KUKA KRL program: puntos.src, puntos.dat

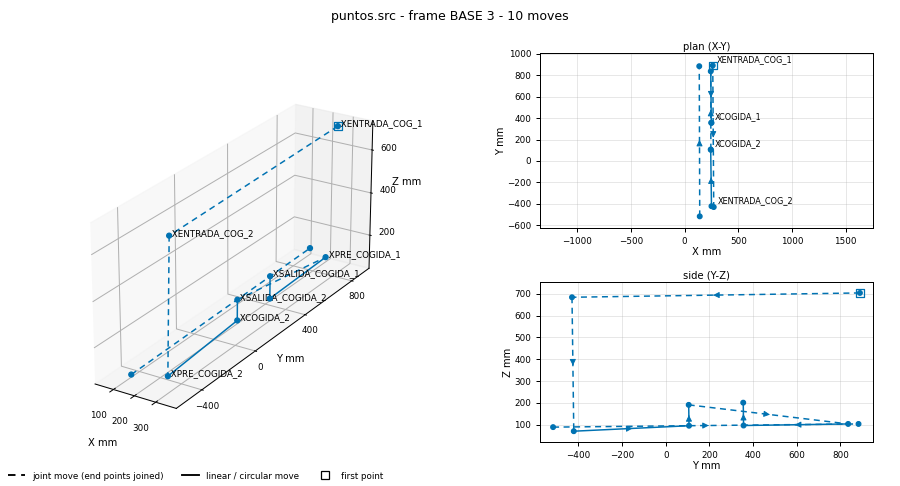
[picture p0: tool path of puntos.src in frame BASE 3, 10 of 13 moves have a stored position in this frame; points joined in program order, loops and branches not executed]
--- puntos.src ---
&ACCESS RVP
&REL 25
&PARAM TEMPLATE = C:\KRC\Roboter\Template\vorgabe
&PARAM EDITMASK = *
DEF PUNTOS( )
;FOLD INI
  ;FOLD BASISTECH INI
    GLOBAL INTERRUPT DECL 3 WHEN $STOPMESS==TRUE DO IR_STOPM ( )
    INTERRUPT ON 3
    BAS (#INITMOV,0 )
  ;ENDFOLD (BASISTECH INI)
  ;FOLD USER INI
    ;Make your modifications here

  ;ENDFOLD (USER INI)
;ENDFOLD (INI)


;FOLD PTP HOME Vel=100 % PDAT6;%{PE}%R 5.6.16,%MKUKATPBASIS,%CMOVE,%VPTP,%P 1:PTP, 2:HOME, 3:, 5:100, 7:PDAT6
$BWDSTART=FALSE
PDAT_ACT=PPDAT6
FDAT_ACT=FHOME
BAS(#PTP_PARAMS,100)
$H_POS=XHOME
PTP XHOME
;ENDFOLD


;FOLD PTP ENTRADA_COG_1 Vel=100 % PDAT1 Tool[2]:MORDAZA Base[3]:TRANSPORTADOR;%{PE}%R 5.6.16,%MKUKATPBASIS,%CMOVE,%VPTP,%P 1:PTP, 2:ENTRADA_COG_1, 3:, 5:100, 7:PDAT1
$BWDSTART=FALSE
PDAT_ACT=PPDAT1
FDAT_ACT=FENTRADA_COG_1
BAS(#PTP_PARAMS,100)
PTP XENTRADA_COG_1
;ENDFOLD


;FOLD PTP ENTRADA_COG_2 Vel=100 % PDAT2 Tool[2]:MORDAZA Base[3]:TRANSPORTADOR;%{PE}%R 5.6.16,%MKUKATPBASIS,%CMOVE,%VPTP,%P 1:PTP, 2:ENTRADA_COG_2, 3:, 5:100, 7:PDAT2
$BWDSTART=FALSE
PDAT_ACT=PPDAT2
FDAT_ACT=FENTRADA_COG_2
BAS(#PTP_PARAMS,100)
PTP XENTRADA_COG_2
;ENDFOLD


;FOLD PTP PRE_COGIDA_2 Vel=100 % PDAT3 Tool[2]:MORDAZA Base[3]:TRANSPORTADOR;%{PE}%R 5.6.16,%MKUKATPBASIS,%CMOVE,%VPTP,%P 1:PTP, 2:PRE_COGIDA_2, 3:, 5:100, 7:PDAT3
$BWDSTART=FALSE
PDAT_ACT=PPDAT3
FDAT_ACT=FPRE_COGIDA_2
BAS(#PTP_PARAMS,100)
PTP XPRE_COGIDA_2
;ENDFOLD


;FOLD LIN COGIDA_2 Vel=2 m/s CPDAT1 Tool[2]:MORDAZA Base[3]:TRANSPORTADOR;%{PE}%R 5.6.16,%MKUKATPBASIS,%CMOVE,%VLIN,%P 1:LIN, 2:COGIDA_2, 3:, 5:2, 7:CPDAT1
$BWDSTART=FALSE
LDAT_ACT=LCPDAT1
FDAT_ACT=FCOGIDA_2
BAS(#CP_PARAMS,2)
LIN XCOGIDA_2
;ENDFOLD


;FOLD LIN SALIDA_COGIDA_2 Vel=2 m/s CPDAT2 Tool[2]:MORDAZA Base[3]:TRANSPORTADOR;%{PE}%R 5.6.16,%MKUKATPBASIS,%CMOVE,%VLIN,%P 1:LIN, 2:SALIDA_COGIDA_2, 3:, 5:2, 7:CPDAT2
$BWDSTART=FALSE
LDAT_ACT=LCPDAT2
FDAT_ACT=FSALIDA_COGIDA_2
BAS(#CP_PARAMS,2)
LIN XSALIDA_COGIDA_2
;ENDFOLD



;FOLD PTP PRE_COGIDA_1 Vel=100 % PDAT4 Tool[2]:MORDAZA Base[3]:TRANSPORTADOR;%{PE}%R 5.6.16,%MKUKATPBASIS,%CMOVE,%VPTP,%P 1:PTP, 2:PRE_COGIDA_1, 3:, 5:100, 7:PDAT4
$BWDSTART=FALSE
PDAT_ACT=PPDAT4
FDAT_ACT=FPRE_COGIDA_1
BAS(#PTP_PARAMS,100)
PTP XPRE_COGIDA_1
;ENDFOLD


;FOLD LIN COGIDA_1 Vel=2 m/s CPDAT3 Tool[2]:MORDAZA Base[3]:TRANSPORTADOR;%{PE}%R 5.6.16,%MKUKATPBASIS,%CMOVE,%VLIN,%P 1:LIN, 2:COGIDA_1, 3:, 5:2, 7:CPDAT3
$BWDSTART=FALSE
LDAT_ACT=LCPDAT3
FDAT_ACT=FCOGIDA_1
BAS(#CP_PARAMS,2)
LIN XCOGIDA_1
;ENDFOLD


;FOLD LIN SALIDA_COGIDA_1 Vel=2 m/s CPDAT4 Tool[2]:MORDAZA Base[3]:TRANSPORTADOR;%{PE}%R 5.6.16,%MKUKATPBASIS,%CMOVE,%VLIN,%P 1:LIN, 2:SALIDA_COGIDA_1, 3:, 5:2, 7:CPDAT4
$BWDSTART=FALSE
LDAT_ACT=LCPDAT4
FDAT_ACT=FSALIDA_COGIDA_1
BAS(#CP_PARAMS,2)
LIN XSALIDA_COGIDA_1
;ENDFOLD



;FOLD PTP DEJA_DARSENA_2 Vel=100 % PDAT7 Tool[2]:MORDAZA Base[2]:DARSENA1;%{PE}%R 5.6.16,%MKUKATPBASIS,%CMOVE,%VPTP,%P 1:PTP, 2:DEJA_DARSENA_2, 3:, 5:100, 7:PDAT7
$BWDSTART=FALSE
PDAT_ACT=PPDAT7
FDAT_ACT=FDEJA_DARSENA_2
BAS(#PTP_PARAMS,100)
PTP XDEJA_DARSENA_2
;ENDFOLD


;FOLD PTP DEJA_DARSENA_1 Vel=100 % PDAT8 Tool[2]:MORDAZA Base[1]:DARSENA1;%{PE}%R 5.6.16,%MKUKATPBASIS,%CMOVE,%VPTP,%P 1:PTP, 2:DEJA_DARSENA_1, 3:, 5:100, 7:PDAT8
$BWDSTART=FALSE
PDAT_ACT=PPDAT8
FDAT_ACT=FDEJA_DARSENA_1
BAS(#PTP_PARAMS,100)
PTP XDEJA_DARSENA_1
;ENDFOLD


;FOLD PTP cog_desplazada Vel=100 % PDAT9 Tool[2]:MORDAZA Base[3]:TRANSPORTADOR;%{PE}%R 5.6.16,%MKUKATPBASIS,%CMOVE,%VPTP,%P 1:PTP, 2:cog_desplazada, 3:, 5:100, 7:PDAT9
$BWDSTART=FALSE
PDAT_ACT=PPDAT9
FDAT_ACT=Fcog_desplazada
BAS(#PTP_PARAMS,100)
PTP Xcog_desplazada
;ENDFOLD

;FOLD PTP cog_desplazada1 Vel=100 % PDAT10 Tool[2]:MORDAZA Base[3]:TRANSPORTADOR;%{PE}%R 5.6.16,%MKUKATPBASIS,%CMOVE,%VPTP,%P 1:PTP, 2:cog_desplazada1, 3:, 5:100, 7:PDAT10
$BWDSTART=FALSE
PDAT_ACT=PPDAT10
FDAT_ACT=Fcog_desplazada1
BAS(#PTP_PARAMS,100)
PTP Xcog_desplazada1
;ENDFOLD
END

--- puntos.dat ---
&ACCESS RVP
&REL 25
&PARAM TEMPLATE = C:\KRC\Roboter\Template\vorgabe
&PARAM EDITMASK = *
DEFDAT  PUNTOS
;FOLD EXTERNAL DECLARATIONS;%{PE}%MKUKATPBASIS,%CEXT,%VCOMMON,%P
;FOLD BASISTECH EXT;%{PE}%MKUKATPBASIS,%CEXT,%VEXT,%P
EXT  BAS (BAS_COMMAND  :IN,REAL  :IN )
DECL INT SUCCESS
;ENDFOLD (BASISTECH EXT)
;FOLD USER EXT;%{E}%MKUKATPUSER,%CEXT,%VEXT,%P
;Make here your modifications

;ENDFOLD (USER EXT)
;ENDFOLD (EXTERNAL DECLARATIONS)
DECL BASIS_SUGG_T LAST_BASIS={POINT1[] "cog_desplazada1         ",POINT2[] "cog_desplazada1         ",CP_PARAMS[] "CPDAT3                  ",PTP_PARAMS[] "PDAT10                  ",CONT[] "                        ",CP_VEL[] "2                       ",PTP_VEL[] "100                     ",SYNC_PARAMS[] "SYNCDAT                 ",SPL_NAME[] "S0                      "}
DECL INT LAST_XP_POINT=0
DECL E6POS XP1={X 267.31131,Y 380.834595,Z 696.146973,A 1.043558,B 1.65328801,C 179.309006,S 6,T 59,E1 0.0,E2 0.0,E3 0.0,E4 0.0,E5 0.0,E6 0.0}
DECL FDAT FP1={TOOL_NO 2,BASE_NO 3,IPO_FRAME #BASE,POINT2[] " ",TQ_STATE FALSE}
DECL PDAT PPDAT1={VEL 100.0,ACC 100.0,APO_DIST 100.0}
DECL E6POS XENTRADA_COG_1={X 262.194702,Y 889.154297,Z 703.763123,A 1.04380703,B 1.65313005,C 179.308701,S 6,T 59,E1 0.0,E2 0.0,E3 0.0,E4 0.0,E5 0.0,E6 0.0}
DECL FDAT FENTRADA_COG_1={TOOL_NO 2,BASE_NO 3,IPO_FRAME #BASE,POINT2[] " ",TQ_STATE FALSE}
DECL E6POS XENTRADA_COG_2={X 271.395813,Y -429.303406,Z 684.026123,A -179.392303,B -0.702468276,C 177.581406,S 6,T 58,E1 0.0,E2 0.0,E3 0.0,E4 0.0,E5 0.0,E6 0.0}
DECL FDAT FENTRADA_COG_2={TOOL_NO 2,BASE_NO 3,IPO_FRAME #BASE,POINT2[] " ",TQ_STATE FALSE}
DECL PDAT PPDAT2={VEL 100.0,ACC 100.0,APO_DIST 100.0}
DECL E6POS XPRE_COGIDA_2={X 250.341797,Y -421.146606,Z 70.6304703,A -179.406097,B -0.698902726,C 177.583694,S 6,T 58,E1 0.0,E2 0.0,E3 0.0,E4 0.0,E5 0.0,E6 0.0}
DECL FDAT FPRE_COGIDA_2={TOOL_NO 2,BASE_NO 3,IPO_FRAME #BASE,POINT2[] " ",TQ_STATE FALSE}
DECL PDAT PPDAT3={VEL 100.0,ACC 100.0,APO_DIST 100.0}
DECL E6POS XCOGIDA_2={X 243.027893,Y 106.545097,Z 95.6698608,A -179.409698,B -0.446659297,C 177.583603,S 6,T 59,E1 0.0,E2 0.0,E3 0.0,E4 0.0,E5 0.0,E6 0.0}
DECL FDAT FCOGIDA_2={TOOL_NO 2,BASE_NO 3,IPO_FRAME #BASE,POINT2[] " ",TQ_STATE FALSE}
DECL LDAT LCPDAT1={VEL 2.0,ACC 100.0,APO_DIST 100.0,APO_FAC 50.0,ORI_TYP #VAR,CIRC_TYP #BASE,JERK_FAC 50.0,EXAX_IGN 0}
DECL E6POS XSALIDA_COGIDA_2={X 244.591003,Y 105.128998,Z 191.241806,A -179.409607,B -0.445713311,C 177.583603,S 6,T 59,E1 0.0,E2 0.0,E3 0.0,E4 0.0,E5 0.0,E6 0.0}
DECL FDAT FSALIDA_COGIDA_2={TOOL_NO 2,BASE_NO 3,IPO_FRAME #BASE,POINT2[] " ",TQ_STATE FALSE}
DECL LDAT LCPDAT2={VEL 2.0,ACC 100.0,APO_DIST 100.0,APO_FAC 50.0,ORI_TYP #VAR,CIRC_TYP #BASE,JERK_FAC 50.0,EXAX_IGN 0}
DECL E6POS XPRE_COGIDA_1={X 243.595703,Y 835.349121,Z 103.8489,A 0.0495731011,B 0.864072084,C 179.297302,S 6,T 59,E1 0.0,E2 0.0,E3 0.0,E4 0.0,E5 0.0,E6 0.0}
DECL FDAT FPRE_COGIDA_1={TOOL_NO 2,BASE_NO 3,IPO_FRAME #BASE,POINT2[] " ",TQ_STATE FALSE}
DECL PDAT PPDAT4={VEL 100.0,ACC 100.0,APO_DIST 100.0}
DECL LDAT LCPDAT3={VEL 2.0,ACC 100.0,APO_DIST 100.0,APO_FAC 50.0,ORI_TYP #VAR,CIRC_TYP #BASE,JERK_FAC 50.0,EXAX_IGN 0}
DECL E6POS XSALIDA_COGIDA_1={X 250.127594,Y 354.823212,Z 201.312805,A 0.05084325,B 0.863396585,C 179.2966,S 6,T 59,E1 0.0,E2 0.0,E3 0.0,E4 0.0,E5 0.0,E6 0.0}
DECL FDAT FSALIDA_COGIDA_1={TOOL_NO 2,BASE_NO 3,IPO_FRAME #BASE,POINT2[] " ",TQ_STATE FALSE}
DECL PDAT PPDAT5={VEL 100.0,ACC 100.0,APO_DIST 100.0}
DECL E6POS XCOGIDA_1={X 248.395905,Y 356.371399,Z 96.664299,A 0.0506648198,B 0.865561903,C 179.296402,S 6,T 59,E1 0.0,E2 0.0,E3 0.0,E4 0.0,E5 0.0,E6 0.0}
DECL FDAT FCOGIDA_1={TOOL_NO 2,BASE_NO 3,IPO_FRAME #BASE,POINT2[] " ",TQ_STATE FALSE}
DECL LDAT LCPDAT4={VEL 2.0,ACC 100.0,APO_DIST 100.0,APO_FAC 50.0,ORI_TYP #VAR,CIRC_TYP #BASE,JERK_FAC 50.0,EXAX_IGN 0}
DECL PDAT PPDAT6={VEL 100.0,ACC 100.0,APO_DIST 100.0}
DECL E6POS XDEJA_DARSENA_2={X 472.251404,Y 536.638611,Z 1677.92395,A 2.64791489,B -0.94016403,C -179.731293,S 6,T 58,E1 0.0,E2 0.0,E3 0.0,E4 0.0,E5 0.0,E6 0.0}
DECL FDAT FDEJA_DARSENA_2={TOOL_NO 2,BASE_NO 2,IPO_FRAME #BASE,POINT2[] " ",TQ_STATE FALSE}
DECL PDAT PPDAT7={VEL 100.0,ACC 100.0,APO_DIST 100.0}
DECL E6POS XDEJA_DARSENA_1={X 443.362091,Y 524.906006,Z -1681.51501,A 179.377808,B 0.200357795,C 0.378010988,S 6,T 58,E1 0.0,E2 0.0,E3 0.0,E4 0.0,E5 0.0,E6 0.0}
DECL FDAT FDEJA_DARSENA_1={TOOL_NO 2,BASE_NO 1,IPO_FRAME #BASE,POINT2[] " ",TQ_STATE FALSE}
DECL PDAT PPDAT8={VEL 100.0,ACC 100.0,APO_DIST 100.0}
DECL E6POS XCOG_DESPLAZADA={X 140.906494,Y -515.904785,Z 89.2991791,A -179.406601,B -0.701284826,C 177.582703,S 6,T 58,E1 0.0,E2 0.0,E3 0.0,E4 0.0,E5 0.0,E6 0.0}
DECL FDAT Fcog_desplazada={TOOL_NO 2,BASE_NO 3,IPO_FRAME #BASE,POINT2[] " ",TQ_STATE FALSE}
DECL PDAT PPDAT9={VEL 100.0,ACC 100.0,APO_DIST 100.0}
DECL E6POS XCOG_DESPLAZADA1={X 136.471603,Y 882.782288,Z 103.830803,A 0.0496506989,B 0.863984823,C 179.297394,S 6,T 59,E1 0.0,E2 0.0,E3 0.0,E4 0.0,E5 0.0,E6 0.0}
DECL FDAT Fcog_desplazada1={TOOL_NO 2,BASE_NO 3,IPO_FRAME #BASE,POINT2[] " ",TQ_STATE FALSE}
DECL PDAT PPDAT10={VEL 100.0,ACC 100.0,APO_DIST 100.0}
ENDDAT
